(* CODESYS project IA_Lab-7.1.project

Project tree, tasks and I/O mapping:
  CAM tables/
  CNC programs/
  Data types/
  Global Variables/
    global variables Global_Variables
    global variables Variable_Configuration
  POUs/
    program PLC_PRG [LD]
  Visualizations/
  GlobalImagePool
*)

// Global Variables/Global_Variables
VAR_GLOBAL
END_VAR

// Global Variables/Variable_Configuration
VAR_CONFIG
END_VAR

// POUs/PLC_PRG
PROGRAM PLC_PRG
VAR
	A: BOOL;
	kjk: TIME;
	L: BOOL;
	T1: TON;
	B: BOOL;
	T2: TP;
	klk: TIME;
	L2: BOOL;
END_VAR

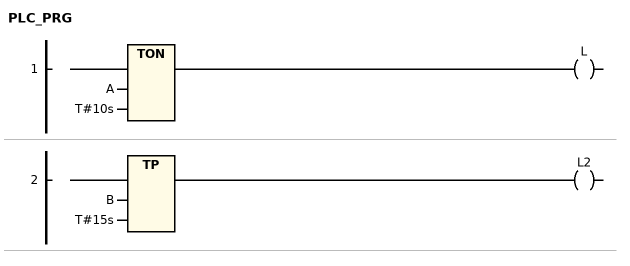
// NETWORK 1
L := TON(A, T#10s);

// NETWORK 2
L2 := TP(B, T#15s);

END_PROGRAM
